TYPE Vec5di : ARRAY[1..5] OF DINT; END_TYPE

(* stored: Version 1.1.0.1, ProductVersion 3.1.4024.11
   DUT Vec5di: Id {d230fc77-25e4-4a02-b0c8-d485112ebc90} *)
